// Code généré automatiquement : NE PAS MODIFIER
FUNCTION CheckDivDInt : DINT
VAR_INPUT
	divisor:DINT;
END_VAR

// Code généré automatiquement : Il s’agit d’une proposition d’implémentation.
{noflow}
IF divisor = 0 THEN
	CheckDivDInt:=1;
ELSE
	CheckDivDInt:=divisor;
END_IF;
{flow}

END_FUNCTION

(* stored: Version 1.1.0.1, ProductVersion 3.1.4024.6
   POU CheckDivDInt: Id {34afacdd-c40c-4236-9a88-2fcfc46e6473}, SpecialFunc CheckDivInt32 *)
